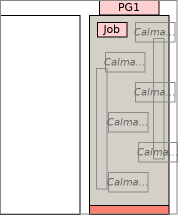
VISUALIZATION _VISU_PmEnable_1Worker  // 178x215
VAR_IN_OUT
  mInst : FB_PrintModule_Base;
END_VAR
    RoundedRectangle (0,15 80x200)
    RoundedRectangle (89,15 80x200), tooltip "WorkerPrint enable"
        toggle mInst.fbWorkerPrint[1]._bEnable
    RoundedRectangle (99,0 60x15), "PG1", tooltip "PG enable"
        toggle mInst.fbWorkerPrint[1]._pAdsPg^.stAds.bI_Enable
    Frame (153,38 11x121)
        shows CalmarCompPrint._VISU_PC_MiniVertical(mInst := mInst._pPc[1]^)
    Frame (96,68 11x121)
        shows CalmarCompPrint._VISU_PC_MiniVertical(mInst := mInst._pPc[2]^)
    Frame (135,22 40x20)
        shows CalmarCompPrint._VISU_PH_TinyVertical(mInst := mInst._pPh[1]^)
    Frame (105,52 40x20)
        shows CalmarCompPrint._VISU_PH_TinyVertical(mInst := mInst._pPh[2]^)
    Frame (135,82 40x20)
        shows CalmarCompPrint._VISU_PH_TinyVertical(mInst := mInst._pPh[3]^)
    Frame (108,112 40x20)
        shows CalmarCompPrint._VISU_PH_TinyVertical(mInst := mInst._pPh[4]^)
    Frame (138,142 40x20)
        shows CalmarCompPrint._VISU_PH_TinyVertical(mInst := mInst._pPh[5]^)
    Frame (108,172 40x20)
        shows CalmarCompPrint._VISU_PH_TinyVertical(mInst := mInst._pPh[6]^)
    RoundedRectangle (97,22 30x15), "Job", tooltip "Job is active", colour toggle: mInst.fbWorkerPrint[1]._bJobActive
    RoundedRectangle (89,205 80x10), tooltip "Worker PrintEnable"
        toggle mInst.fbWorkerPrint[1].bWorkerPrintEnable
END_VISUALIZATION

(* stored: Version 1.1.0.1, ProductVersion 3.1.4024.11
   Visu _VISU_PmEnable_1Worker: Id {64e5fb99-bdde-46c9-9494-19b5a659f034} *)
